HMI tags "Default tag table"
   "Screen" : UInt, internal
   "OPPovely_P12 Nahoru" : Bool = PLC OPPovely."P12 Nahoru" AT %DB20.DBX1.5, 1 s
   "OPPovely_P12 Dolu" : Bool = PLC OPPovely."P12 Dolu" AT %DB20.DBX1.6, 1 s
   "Počítadlo_DB_Linka1.Požadovaný počet vrstev" : Int = PLC Počítadlo_DB.Linka1."Požadovaný počet vrstev" AT %DB15.DBW0, 1 s
   "Počítadlo_DB_Linka1.Aktuální počet vrstev" : Int = PLC Počítadlo_DB.Linka1."Aktuální počet vrstev" AT %DB15.DBW2, 1 s
   "Počítadlo_DB_Linka1.Aktuální počet půlvrstev" : Int = PLC Počítadlo_DB.Linka1."Aktuální počet půlvrstev" AT %DB15.DBW4, 1 s
   "Počítadlo_DB_Linka2.Požadovaný počet vrstev" : Int = PLC Počítadlo_DB.Linka2."Požadovaný počet vrstev" AT %DB15.DBW6, 1 s
   "Počítadlo_DB_Linka2.Aktuální počet vrstev" : Int = PLC Počítadlo_DB.Linka2."Aktuální počet vrstev" AT %DB15.DBW8, 1 s
   "Počítadlo_DB_Linka2.Aktuální počet půlvrstev" : Int = PLC Počítadlo_DB.Linka2."Aktuální počet půlvrstev" AT %DB15.DBW10, 1 s
   "OPPovely_P3 Start" : Bool = PLC OPPovely."P3 Start" AT %DB20.DBX0.3, 1 s
   "OPPovely_P4 Start" : Bool = PLC OPPovely."P4 Start" AT %DB20.DBX0.4, 1 s
   "OPPovely_P5 Start" : Bool = PLC OPPovely."P5 Start" AT %DB20.DBX0.5, 1 s
   "OPPovely_Destohovač ramena sevřít" : Bool = PLC OPPovely."Destohovač ramena sevřít" AT %DB20.DBX1.0, 1 s
   "OPPovely_Destohovač dolu" : Bool = PLC OPPovely."Destohovač dolu" AT %DB20.DBX0.7, 1 s
   "OPPovely_Destohovač nahoru" : Bool = PLC OPPovely."Destohovač nahoru" AT %DB20.DBX0.6, 1 s
   "OPPovely_P8 Start" : Bool = PLC OPPovely."P8 Start" AT %DB20.DBX1.2, 1 s
   "OPPovely_P12 Start" : Bool = PLC OPPovely."P12 Start" AT %DB20.DBX1.3, 1 s
   "OPPovely_P11 Start" : Bool = PLC OPPovely."P11 Start" AT %DB20.DBX2.0, 1 s
   "OPPovely_P11 Nahoru" : Bool = PLC OPPovely."P11 Nahoru" AT %DB20.DBX2.2, 1 s
   "OPPovely_P11 Dolu" : Bool = PLC OPPovely."P11 Dolu" AT %DB20.DBX2.3, 1 s
   "OPPovely_P12 Vzad" : Bool = PLC OPPovely."P12 Vzad" AT %DB20.DBX1.4, 1 s
   "OPPovely_P11 Vzad" : Bool = PLC OPPovely."P11 Vzad" AT %DB20.DBX2.1, 1 s
   "OPPovely_P17 Start" : Bool = PLC OPPovely."P17 Start" AT %DB20.DBX2.5, 1 s
   "OPPovely_P18 Start" : Bool = PLC OPPovely."P18 Start" AT %DB20.DBX2.6, 1 s
   "OPPovely_P19 Ovíječka Start" : Bool = PLC OPPovely."P19 Ovíječka Start" AT %DB20.DBX2.7, 1 s
   "OPPovely_P20 Start" : Bool = PLC OPPovely."P20 Start" AT %DB20.DBX3.0, 1 s
   "OPPovely_P21 Start" : Bool = PLC OPPovely."P21 Start" AT %DB20.DBX3.1, 1 s
   "OPPovely_OP Start" : Bool = PLC OPPovely."OP Start" AT %DB20.DBX0.0, 1 s
   "OPPovely_OP Manual" : Bool = PLC OPPovely."OP Manual" AT %DB20.DBX0.2, 1 s
   "Globální řízení_DB_Automat" : Bool = PLC "Globální řízení_DB".Automat AT %DB12.DBX0.0, 1 s
   "Rovnání palety P12 sevřít" : Bool = PLC "Rovnání palety P12 sevřít" AT %Q47.5, 1 s
   "OPPovely_P11 Rovnání" : Bool = PLC OPPovely."P11 Rovnání" AT %DB20.DBX2.4, 1 s
   "OPPovely_P12 Rovnání" : Bool = PLC OPPovely."P12 Rovnání" AT %DB20.DBX1.7, 1 s
   "Destohovač sevřít" : Bool = PLC "Destohovač sevřít" AT %Q41.7, 1 s
   "OPPovely_Linka1.P49 Start" : Bool = PLC OPPovely.Linka1."P49 Start" AT %DB20.DBX5.5, 1 s
   "OPPovely_Linka1.P47.1 Start" : Bool = PLC OPPovely.Linka1."P47.1 Start" AT %DB20.DBX5.1, 1 s
   "OPPovely_Linka1.P47.2 Start" : Bool = PLC OPPovely.Linka1."P47.2 Start" AT %DB20.DBX5.3, 1 s
   "OPPovely_Linka1.P37 Start" : Bool = PLC OPPovely.Linka1."P37 Start" AT %DB20.DBX5.0, 1 s
   "OPPovely_Linka1.P35 Elevátor Start" : Bool = PLC OPPovely.Linka1."P35 Elevátor Start" AT %DB20.DBX4.7, 1 s
   "OPPovely_Linka1.P36 Start" : Bool = PLC OPPovely.Linka1."P36 Start" AT %DB20.DBX4.6, 1 s
   "OPPovely_Linka1.P33 Start" : Bool = PLC OPPovely.Linka1."P33 Start" AT %DB20.DBX4.4, 1 s
   "OPPovely_Linka1.P29 Start" : Bool = PLC OPPovely.Linka1."P29 Start" AT %DB20.DBX4.3, 1 s
   "OPPovely_Linka1.P27 Elevátor Start" : Bool = PLC OPPovely.Linka1."P27 Elevátor Start" AT %DB20.DBX4.2, 1 s
   "OPPovely_Linka1.P28 Start" : Bool = PLC OPPovely.Linka1."P28 Start" AT %DB20.DBX4.1, 1 s
   "OPPovely_Linka1.P23 Start" : Bool = PLC OPPovely.Linka1."P23 Start" AT %DB20.DBX4.0, 1 s
   "OPPovely_Linka1.Klapka P47.1" : Bool = PLC OPPovely.Linka1."Klapka P47.1" AT %DB20.DBX5.2, 1 s
   "OPPovely_Linka1.Klapka P47.2" : Bool = PLC OPPovely.Linka1."Klapka P47.2" AT %DB20.DBX5.4, 1 s
   "OPPovely_Linka1.Klapka P33" : Bool = PLC OPPovely.Linka1."Klapka P33" AT %DB20.DBX4.5, 1 s
   "Klapka 47.2 nahoru" : Bool = PLC "Klapka 47.2 nahoru" AT %Q46.2, 1 s
   "Klapka P47.1 nahoru" : Bool = PLC "Klapka P47.1 nahoru" AT %Q46.0, 1 s
   "Klapka P33 nahoru" : Bool = PLC "Klapka P33 nahoru" AT %Q46.4, 1 s
   "Rovnání palety P11 sevřít" : Bool = PLC "Rovnání palety P11 sevřít" AT %Q47.1, 1 s

HMI tags "Errors"
   "Errors 1" : Int AT %DB100.DBW2, 1 s
   "Evaluated errors 1" : Int AT %DB100.DBW4, 1 s

discrete alarms
   1: 'Central stop / Nouzové zastavení', class Chyby, trigger "Errors 1" bit 8
   2: 'Vypnuty silové obvody', class Chyby, trigger "Errors 1" bit 9
   3: 'Nízký tlak vzduchu', class Chyby, trigger "Errors 1" bit 10
   4: 'Jistič doptavníku P1', class Chyby, trigger "Errors 1" bit 11
   5: 'Jistič dopravníku P2 nebo P3', class Chyby, trigger "Errors 1" bit 12
   6: 'Jističe válcovačky nebo dopravníku ovíječky', class Chyby, trigger "Errors 1" bit 13
   7: 'reserva', class Chyby, trigger "Errors 1" bit 14
   8: 'Porucha bezpečnostního relé', class Chyby, trigger "Errors 1" bit 15
   9: 'reserva_1', class Chyby, trigger "Errors 1" bit 0
   10: 'reserva_1_1', class Chyby, trigger "Errors 1" bit 1
   11: 'reserva_2', class Chyby, trigger "Errors 1" bit 2
   12: 'reserva_2_1', class Chyby, trigger "Errors 1" bit 3
   13: 'reserva_3', class Chyby, trigger "Errors 1" bit 4
   14: 'reserva_3_1', class Chyby, trigger "Errors 1" bit 5
   15: 'reserva_3_2', class Chyby, trigger "Errors 1" bit 6
   16: 'reserva_3_3', class Chyby, trigger "Errors 1" bit 7

text list "Destohovač ramena": 0 '►◄'; 1 '◄►'

text list "Poloha rovnání": 0 '▼'; 1 '▲'

text list "Poloha klapky": 0 '▲'; 1 '▼'

graphic list "Graphic_list_1": 0 'play-512'; 1 'Stop_button_play_pause_music'

screen "Root screen" 320x240, template "Template_1"
   on GenerateScreen: SetTag("Screen", 1)
   IOField "I/O field_1" at 270,138 size 30x23; FormatPattern 9
      ProcessValue <- "Počítadlo_DB_Linka1.Aktuální počet vrstev"
   IOField "I/O field_2" at 8,168 size 30x23; FormatPattern 99
      ProcessValue <- "Počítadlo_DB_Linka2.Aktuální počet půlvrstev"
   TextField "Text field_1" at 95,138 size 127x13; Text 'Aktuální počet pytlů: / Aktuální počet půlvrstev:'
   TextField "Text field_2" at 71,171 size 175x13; Text 'Aktuální počet vrstev: / Aktuální počet kompletních vrstev:'
   IOField "I/O field_3" at 8,104 size 30x23; FormatPattern 99
      ProcessValue <- "Počítadlo_DB_Linka2.Požadovaný počet vrstev"
   TextField "Text field_4" at 100,107 size 117x13; Text 'Počet vrstev na paletě: / Počet vrstev na paletu:'
   IOField "I/O field_5" at 270,170 size 30x23; FormatPattern 99
      ProcessValue <- "Počítadlo_DB_Linka1.Aktuální počet půlvrstev"
   IOField "I/O field_6" at 8,136 size 30x23; FormatPattern 9
      ProcessValue <- "Počítadlo_DB_Linka2.Aktuální počet vrstev"
   IOField "I/O field_7" at 270,106 size 30x23; FormatPattern s99999
      ProcessValue <- "Počítadlo_DB_Linka1.Požadovaný počet vrstev"
   AlarmView "Alarm view_1" at 6,36 size 310x35
   TextField "Text field_3" at 8,80 size 48x13; Text 'LINKA 2:'
   TextField "Text field_5" at 256,80 size 48x13; Text 'LINKA 1:'
   GraphicView "Logo" at 4,5 size 156x31; Picture "logo okraj"

screen "Manual" 320x240
   on GenerateScreen: SetTag("Screen", 2)
   Button "Button_5" at 192,80 size 32x32; TextOff '▲'
      on Press: function_b14e0dd5("OPPovely_Destohovač nahoru", 0)
   Button "Button_7" at 232,96 size 48x24; TextOff 'Dopravník P3 / 1èáéçê'; TextList "Destohovač ramena"
      on Press: function_b14e0dd5("OPPovely_Destohovač ramena sevřít", 0)
      ProcessValue <- "Destohovač sevřít"
   Button "Button_9" at 288,80 size 32x32; TextOff '▼'
      on Press: function_b14e0dd5("OPPovely_Destohovač dolu", 0)
   Button "Button_6" at 232,40 size 48x24; TextOff 'Dopravník P1 ˅ ˅'
      on Press: SetBit("OPPovely_P4 Start")
   Button "Button_3" at 232,72 size 48x24; TextOff 'Dopravník P1 ˅ ˅'
      on Press: function_b14e0dd5("OPPovely_P5 Start", 0)
   Button "Button_2" at 232,9 size 48x24; TextOff 'Dopravník P1 ˅ ˅'
      on Press: function_b14e0dd5("OPPovely_P3 Start", 0)
   Button "Button_8" at 233,127 size 48x69; TextOff 'Dopravník P1 ˅ ˅'
      on Press: function_b14e0dd5("OPPovely_P8 Start", 0)
   Button "Button_10" at 205,129 size 25x32; TextOff 'Dopravník P1 / ˂˂'
      on Press: function_b14e0dd5("OPPovely_P12 Start", 0)
   Button "Button_11" at 64,129 size 28x32; TextOff 'Dopravník P1 / ˃˃'
      on Press: function_b14e0dd5("OPPovely_P12 Vzad", 0)
   Button "Button_12" at 205,164 size 25x32; TextOff 'Dopravník P1 / ˂˂'
      on Press: function_b14e0dd5("OPPovely_P11 Start", 0)
   Button "Button_13" at 64,164 size 28x32; TextOff 'Dopravník P1 / ˃˃'
      on Press: function_b14e0dd5("OPPovely_P11 Vzad", 0)
   Button "Button_4" at 93,129 size 31x32; TextOff 'Dopravník P3 / ▲'
      on Press: function_b14e0dd5("OPPovely_P12 Nahoru", 0)
   Button "Button_14" at 174,129 size 29x32; TextOff 'Dopravník P3 / ▼'
      on Release: ResetBit("OPPovely_P12 Dolu")
      on Press: SetBit("OPPovely_P12 Dolu")
   Button "Button_15" at 12,127 size 48x69; TextOff 'Dopravník P1 ˄ ˄'
      on Press: function_b14e0dd5("OPPovely_P17 Start", 0)
   Button "Button_16" at 94,164 size 31x32; TextOff 'Dopravník P3 / ▲'
      on Press: function_b14e0dd5("OPPovely_P11 Nahoru", 0)
   Button "Button_17" at 174,164 size 29x32; TextOff 'Dopravník P3 / ▼'
      on Press: function_b14e0dd5("OPPovely_P11 Dolu", 0)
   Button "Button_18" at 12,98 size 48x24; TextOff 'Dopravník P1 ˄ ˄'
      on Press: function_b14e0dd5("OPPovely_P18 Start", 0)
   Button "Button_19" at 12,66 size 48x24; TextOff 'Dopravník P1 ˄ ˄'
      on Press: function_b14e0dd5("OPPovely_P19 Ovíječka Start", 0)
   Button "Button_20" at 12,34 size 48x24; TextOff 'Dopravník P1 ˄ ˄'
      on Press: function_b14e0dd5("OPPovely_P20 Start", 0)
   Button "Button_21" at 12,3 size 48x24; TextOff 'Dopravník P1 ˄ ˄'
      on Press: function_b14e0dd5("OPPovely_P21 Start", 0)
   Button "Start screen" at 1,202 size 52x37; TextOn 'Start screen'; TextOff 'Start screen'; PictureOn "NavigateHome_KTP600_Basic_color_PN"; PictureOff "NavigateHome_KTP600_Basic_color_PN"
      on Release: ActivateScreen("Root screen", 0)
   Button "Button_1" at 64,202 size 103x36; TextOff 'Dopravník P1 Dopravníky kartonů LINKA 2'
      on Press: function_b14e0dd5("OPPovely_P3 Start", 0)
   Button "Button_22" at 178,202 size 103x36; TextOff 'Dopravník P1 Dopravníky kartonů LINKA 1'
      on Release: ActivateScreen("Manual_Linka_1", 0)
   Button "Button_23" at 125,129 size 48x32; TextOff 'Dopravník P1 ˄ ˄'; TextList "Poloha rovnání"
      on Press: function_b14e0dd5("OPPovely_P12 Rovnání", 0)
      ProcessValue <- "Rovnání palety P12 sevřít"
   Button "Button_24" at 125,164 size 48x32; TextOff 'Dopravník P1 ˄ ˄'; TextList "Poloha rovnání"
      on Press: function_b14e0dd5("OPPovely_P11 Rovnání", 0)
      ProcessValue <- "Rovnání palety P11 sevřít"

screen "Setting" 320x240, template "Template_1"
   on GenerateScreen: SetTag("Screen", 3)
   Button "Button_1" at 25,60 size 75x28; TextOff 'Login / Přihlášení'
      on Press: function_a2a04561()
   Button "Button_2" at 25,105 size 75x28; TextOff 'Logout / Odhlášení'
      on Press: function_f23ef4c9()
   Button "Button_3" at 165,60 size 96x32; TextOff 'Text'
      on Release: function_ef3f5d25("Alarm window_Unacknowledged", -1)

screen "Alarms" 320x240, template "Template_1"
   AlarmView "Alarm view_1" at 0,41 size 320x151

Template "Template_1" 320x240
   Button "Exit" at 266,202 size 52x37; TextOff 'Exit'; Authorization "User administration"; PictureOff "ExitRuntime_KTP600_Basic_color_PN"; PictureOn "ExitRuntime_KTP600_Basic_color_PN"
      on Release: StopRuntime(0)
   Button "Template_Button" at 213,202 size 52x37; TextOff 'Text'; PictureOff "custom_settings-512"
      on Release: ActivateScreen("Setting", 0)
   Button "Template_Button_1" at 160,202 size 52x37; TextOff 'Text'; PictureOff "Hand-Touch-icon-300x300"
      on Press: function_b14e0dd5("OPPovely_OP Manual", 0)
      on Release: ResetBit("OPPovely_OP Manual"); ActivateScreen("Manual", 0)
   Button "Template_Button_2" at 107,202 size 52x37; TextOff 'Text'; PictureList "Graphic_list_1"
      on Press: function_b14e0dd5("OPPovely_OP Start", 0)
      ProcessValue <- "Globální řízení_DB_Automat"
   Button "Alarms" at 54,202 size 52x37; TextOn 'Alarms'; TextOff 'Alarms'; PictureOn "AlarmDisplay_KTP600_Basic_color_PN"; PictureOff "AlarmDisplay_KTP600_Basic_color_PN"
      on Release: ActivateScreen("Alarms", 0)
   Button "Start screen" at 1,202 size 52x37; TextOn 'Start screen'; TextOff 'Start screen'; PictureOn "NavigateHome_KTP600_Basic_color_PN"; PictureOff "NavigateHome_KTP600_Basic_color_PN"
      on Release: ActivateScreen("Root screen", 0)

screen "Manual_Linka_1" 320x240
   on GenerateScreen: SetTag("Screen", 5)
   Button "Button_13" at 130,208 size 116x26; TextOff 'Dopravník P1 / ˃˃'
      on Press: function_b14e0dd5("OPPovely_Linka1.P33 Start", 0)
   Button "Button_15" at 130,151 size 48x24; TextOff 'Dopravník P1 ˄ -- --˄'
      on Press: function_b14e0dd5("OPPovely_Linka1.P35 Elevátor Start", 0)
   Button "Button_18" at 130,121 size 48x24; TextOff 'Dopravník P1 ˄ ˄'
      on Press: function_b14e0dd5("OPPovely_Linka1.P37 Start", 0)
   Button "Button_19" at 130,36 size 48x24; TextOff 'Dopravník P1 ˄ ˄'
      on Press: function_b14e0dd5("OPPovely_Linka1.P47.2 Start", 0)
   Button "Button_20" at 130,65 size 48x24; TextOff 'Dopravník P1 ˄ ˄'
      on Press: function_b14e0dd5("OPPovely_Linka1.P47.1 Start", 0)
   Button "Button_21" at 130,6 size 48x24; TextOff 'Dopravník P1 ˄ ˄'
      on Press: function_b14e0dd5("OPPovely_Linka1.P49 Start", 0)
   Button "Start screen" at 1,202 size 52x37; TextOn 'Start screen'; TextOff 'Start screen'; PictureOn "NavigateHome_KTP600_Basic_color_PN"; PictureOff "NavigateHome_KTP600_Basic_color_PN"
      on Release: ActivateScreen("Root screen", 0)
   Button "Start screen_1" at 268,200 size 52x37; TextOn 'Start screen'; TextOff 'Start screen'; PictureOn "NavigateHome_KTP600_Basic_color_PN"; PictureOff "Go-back-icon"
      on Release: ActivateScreen("Manual", 0)
   GraphicView "Graphic view_1" at 130,93 size 48x24; Picture "Graphic_10"
   Button "Button_2" at 130,180 size 48x24; TextOff 'Dopravník P1 ˄ ˄'
      on Press: function_b14e0dd5("OPPovely_Linka1.P36 Start", 0)
   Button "Button_1" at 260,34 size 48x24; TextOff 'Dopravník P1 ˄ ˄'
      on Press: function_b14e0dd5("OPPovely_Linka1.P29 Start", 0)
   Button "Button_3" at 260,104 size 48x24; TextOff 'Dopravník P1 ˄ ˄'
      on Press: function_b14e0dd5("OPPovely_Linka1.P28 Start", 0)
   Button "Button_4" at 260,69 size 48x24; TextOff 'Dopravník P1 ˄ -- --˄'
      on Press: function_b14e0dd5("OPPovely_Linka1.P27 Elevátor Start", 0)
   Button "Button_5" at 259,138 size 48x24; TextOff 'Dopravník P1 ˄ ˄'
      on Press: function_b14e0dd5("OPPovely_Linka1.P23 Start", 0)
   Button "Button_6" at 72,65 size 48x24; TextOff 'Dopravník P1 ˄ ˄'; TextList "Poloha klapky"
      on Press: function_b14e0dd5("OPPovely_Linka1.Klapka P47.1", 0)
      ProcessValue <- "Klapka P47.1 nahoru"
   Button "Button_7" at 72,36 size 48x24; TextOff 'Dopravník P1 ˄ ˄'; TextList "Poloha klapky"
      on Press: function_b14e0dd5("OPPovely_Linka1.Klapka P47.2", 0)
      ProcessValue <- "Klapka 47.2 nahoru"
   Button "Button_8" at 75,209 size 48x24; TextOff 'Dopravník P1 ˄ ˄'; TextList "Poloha klapky"
      on Press: function_b14e0dd5("OPPovely_Linka1.Klapka P33", 0)
      ProcessValue <- "Klapka P33 nahoru"
*)